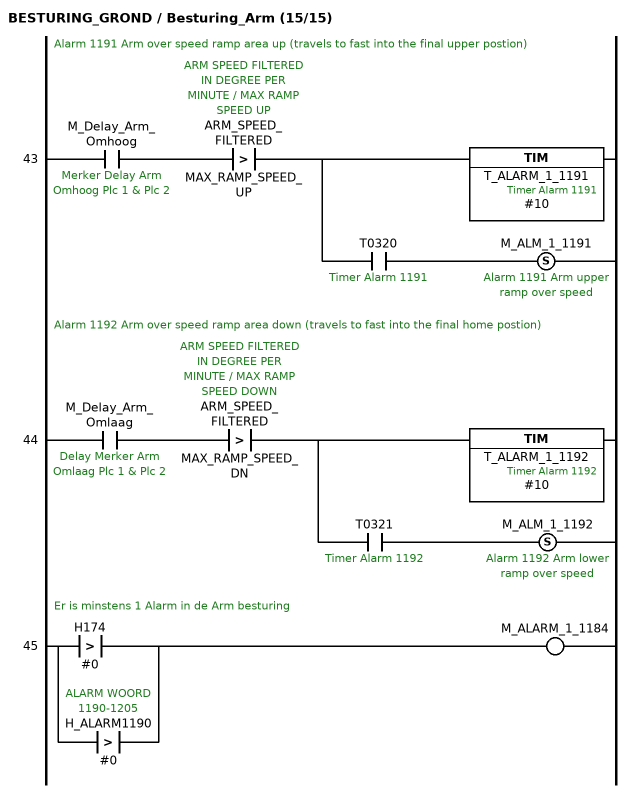
; [picture p168: BESTURING_GROND / Besturing_Arm, rungs 43-45]
; rung 43: Alarm 1191 Arm over speed ramp area up (travels to fast into the final upper postion)
LD M_Delay_Arm_Omhoog  ; Merker Delay Arm Omhoog Plc 1 & Plc 2
AND>F(333) ARM_SPEED_FILTERED MAX_RAMP_SPEED_UP  ; ARM SPEED FILTERED IN DEGREE PER MINUTE, MAX RAMP SPEED UP
TIM T_ALARM_1_1191 #10  ; Timer Alarm 1191
AND T0320  ; Timer Alarm 1191
SET M_ALM_1_1191  ; Alarm 1191 Arm upper ramp over speed
; rung 44: Alarm 1192 Arm over speed ramp area down (travels to fast into the final home postion)
LD M_Delay_Arm_Omlaag  ; Delay Merker Arm Omlaag Plc 1 & Plc 2
AND>F(333) ARM_SPEED_FILTERED MAX_RAMP_SPEED_DN  ; ARM SPEED FILTERED IN DEGREE PER MINUTE, MAX RAMP SPEED DOWN
TIM T_ALARM_1_1192 #10  ; Timer Alarm 1192
AND T0321  ; Timer Alarm 1192
SET M_ALM_1_1192  ; Alarm 1192 Arm lower ramp over speed
; rung 45: Er is minstens 1 Alarm in de Arm besturing
LD>(320) H174 #0
OR>(320) H_ALARM1190 #0  ; ALARM WOORD 1190-1205
OUT M_ALARM_1_1184

### Section Einde_Besturing_Grond
; rung 0
END(001)

## Program SIGNALEN_EILAND (cyclic task 10)

### Section Fast_Counter_Control
; rung 0: adress in 363-365 adrs uit 62-64

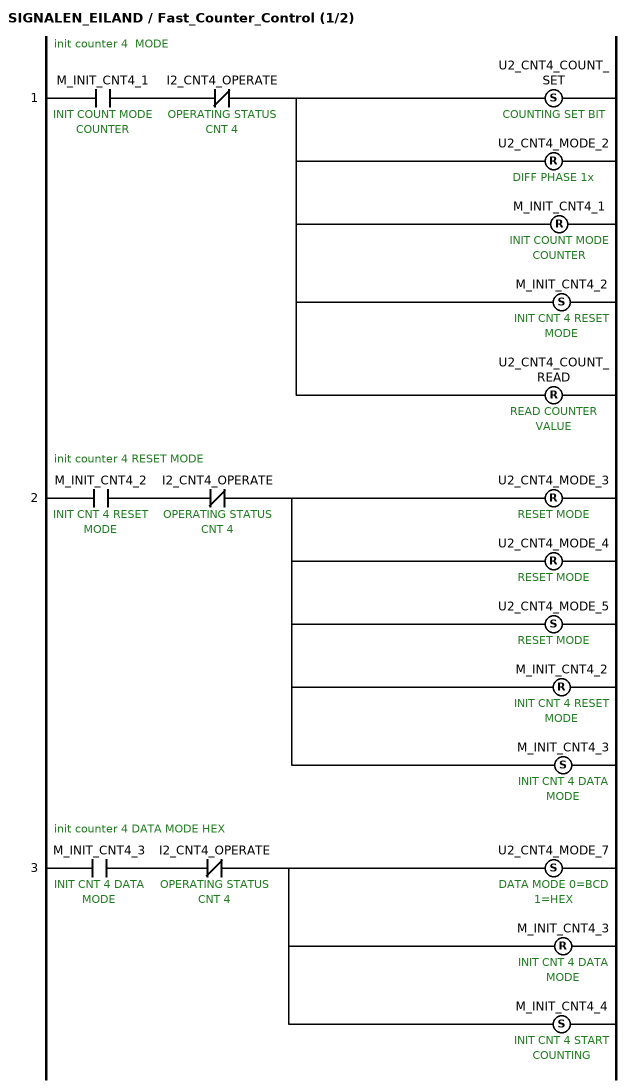
; rung 1: init counter 4  MODE
LD M_INIT_CNT4_1  ; INIT COUNT MODE COUNTER
ANDNOT I2_CNT4_OPERATE  ; OPERATING STATUS CNT 4
SET U2_CNT4_COUNT_SET  ; COUNTING SET BIT
RSET U2_CNT4_MODE_2  ; DIFF PHASE 1x
RSET M_INIT_CNT4_1  ; INIT COUNT MODE COUNTER
SET M_INIT_CNT4_2  ; INIT CNT 4 RESET MODE
RSET U2_CNT4_COUNT_READ  ; READ COUNTER VALUE
; rung 2: init counter 4 RESET MODE
LD M_INIT_CNT4_2  ; INIT CNT 4 RESET MODE
ANDNOT I2_CNT4_OPERATE  ; OPERATING STATUS CNT 4
RSET U2_CNT4_MODE_3  ; RESET MODE
RSET U2_CNT4_MODE_4  ; RESET MODE
SET U2_CNT4_MODE_5  ; RESET MODE
RSET M_INIT_CNT4_2  ; INIT CNT 4 RESET MODE
SET M_INIT_CNT4_3  ; INIT CNT 4 DATA MODE
; rung 3: init counter 4 DATA MODE HEX
LD M_INIT_CNT4_3  ; INIT CNT 4 DATA MODE
ANDNOT I2_CNT4_OPERATE  ; OPERATING STATUS CNT 4
SET U2_CNT4_MODE_7  ; DATA MODE 0=BCD 1=HEX
RSET M_INIT_CNT4_3  ; INIT CNT 4 DATA MODE
SET M_INIT_CNT4_4  ; INIT CNT 4 START COUNTING

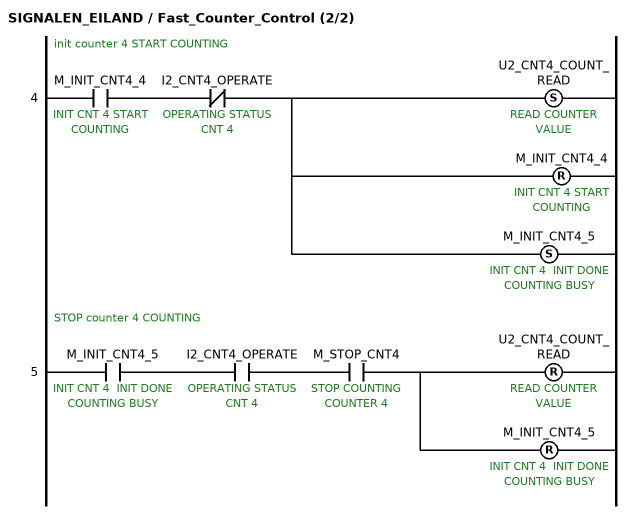
; rung 4: init counter 4 START COUNTING
LD M_INIT_CNT4_4  ; INIT CNT 4 START COUNTING
ANDNOT I2_CNT4_OPERATE  ; OPERATING STATUS CNT 4
SET U2_CNT4_COUNT_READ  ; READ COUNTER VALUE
RSET M_INIT_CNT4_4  ; INIT CNT 4 START COUNTING
SET M_INIT_CNT4_5  ; INIT CNT 4  INIT DONE COUNTING BUSY
; rung 5: STOP counter 4 COUNTING
LD M_INIT_CNT4_5  ; INIT CNT 4  INIT DONE COUNTING BUSY
AND I2_CNT4_OPERATE  ; OPERATING STATUS CNT 4
AND M_STOP_CNT4  ; STOP COUNTING COUNTER 4
RSET U2_CNT4_COUNT_READ  ; READ COUNTER VALUE
RSET M_INIT_CNT4_5  ; INIT CNT 4  INIT DONE COUNTING BUSY

### Section Incremental_Encoder_Decoder_4

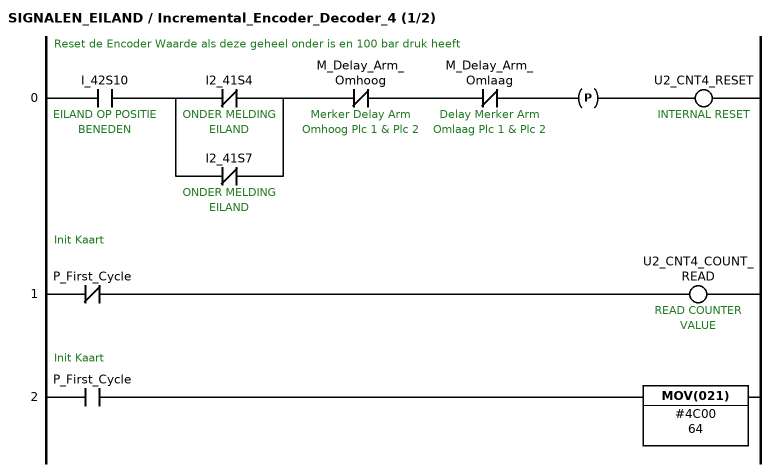
; rung 0: Reset de Encoder Waarde als deze geheel onder is en 100 bar druk heeft
LD I_42S10  ; EILAND OP POSITIE BENEDEN
LDNOT I2_41S4  ; ONDER MELDING EILAND
ORNOT I2_41S7  ; ONDER MELDING EILAND
ANDLD
ANDNOT M_Delay_Arm_Omhoog  ; Merker Delay Arm Omhoog Plc 1 & Plc 2
ANDNOT M_Delay_Arm_Omlaag  ; Delay Merker Arm Omlaag Plc 1 & Plc 2
UP(521)
OUT U2_CNT4_RESET  ; INTERNAL RESET
; rung 1: Init Kaart
LDNOT P_First_Cycle
OUT U2_CNT4_COUNT_READ  ; READ COUNTER VALUE
; rung 2: Init Kaart
LD P_First_Cycle
MOV(021) #4C00 64

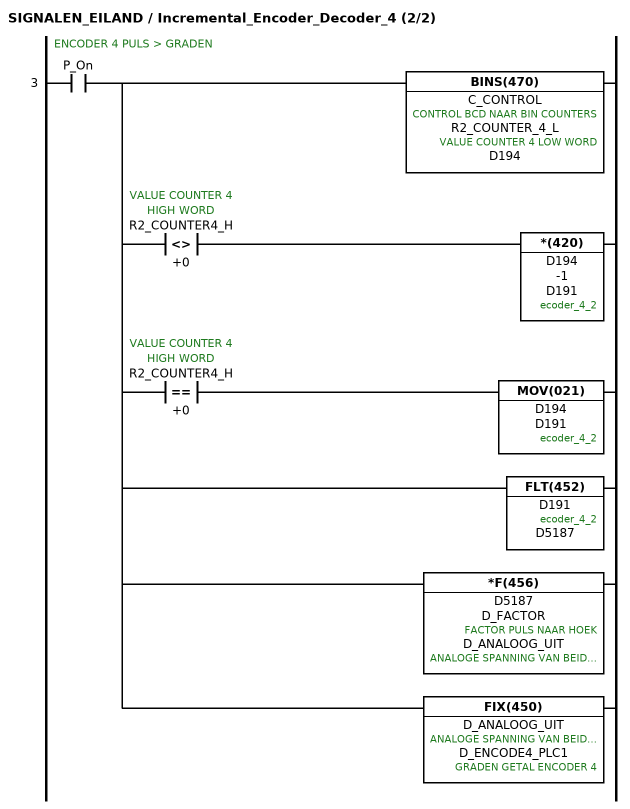
; rung 3: ENCODER 4 PULS > GRADEN
LD P_On
OUT TR0
BINS(470) C_CONTROL R2_COUNTER_4_L D194  ; CONTROL BCD NAAR BIN COUNTERS, VALUE COUNTER 4 LOW WORD
AND<>S(307) R2_COUNTER4_H +0  ; VALUE COUNTER 4 HIGH WORD
*(420) D194 -1 D191  ; ecoder_4_2
LD TR0
AND=S(302) R2_COUNTER4_H +0  ; VALUE COUNTER 4 HIGH WORD
MOV(021) D194 D191  ; ecoder_4_2
LD TR0
FLT(452) D191 D5187  ; ecoder_4_2
*F(456) D5187 D_FACTOR D_ANALOOG_UIT  ; FACTOR PULS NAAR HOEK, ANALOGE SPANNING VAN BEIDE PLC'S
FIX(450) D_ANALOOG_UIT D_ENCODE4_PLC1  ; ANALOGE SPANNING VAN BEIDE PLC'S, GRADEN GETAL ENCODER 4

### Section Horizon_Decoder_Eiland
; rung 0: De Horizon Decoder is alleen aanwezig in Plc 2 Omdat de analoog waarde allen daar binnen word gelezen.

### Section Controle_Positie_Eiland

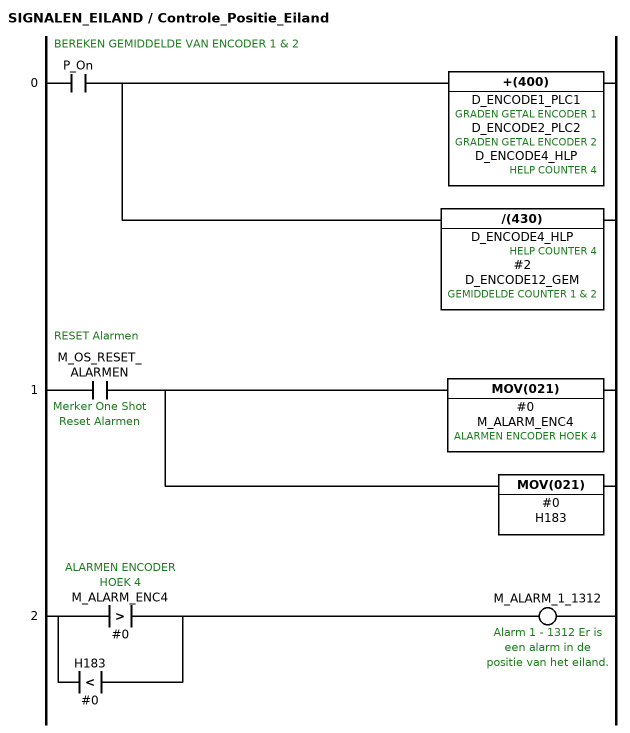
; rung 0: BEREKEN GEMIDDELDE VAN ENCODER 1 & 2
LD P_On
+(400) D_ENCODE1_PLC1 D_ENCODE2_PLC2 D_ENCODE4_HLP  ; GRADEN GETAL ENCODER 1, GRADEN GETAL ENCODER 2, HELP COUNTER 4
/(430) D_ENCODE4_HLP #2 D_ENCODE12_GEM  ; HELP COUNTER 4, GEMIDDELDE COUNTER 1 & 2
; rung 1: RESET Alarmen
LD M_OS_RESET_ALARMEN  ; Merker One Shot Reset Alarmen
MOV(021) #0 M_ALARM_ENC4  ; ALARMEN ENCODER HOEK 4
MOV(021) #0 H183
; rung 2
LD>(320) M_ALARM_ENC4 #0  ; ALARMEN ENCODER HOEK 4
OR<(310) H183 #0
OUT M_ALARM_1_1312  ; Alarm 1 - 1312 Er is een alarm in de positie van het eiland.

### Section Controle_Level_Switches_Eiland

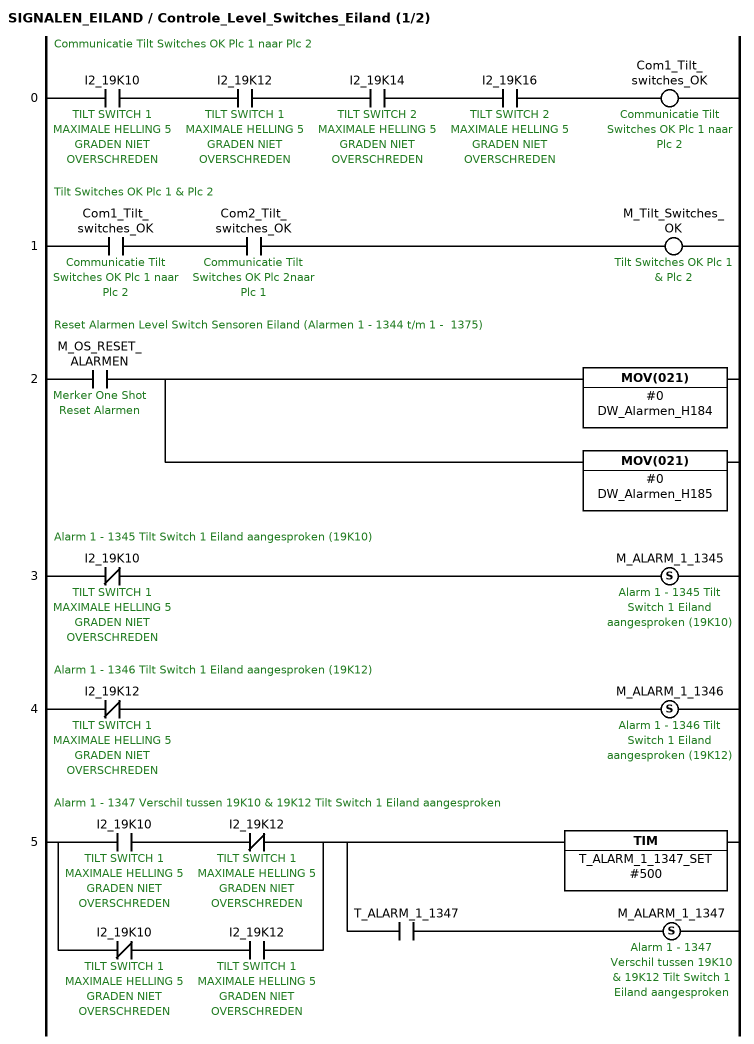
; rung 0: Communicatie Tilt Switches OK Plc 1 naar Plc 2
LD I2_19K10  ; TILT SWITCH 1 MAXIMALE HELLING 5 GRADEN NIET OVERSCHREDEN
AND I2_19K12  ; TILT SWITCH 1 MAXIMALE HELLING 5 GRADEN NIET OVERSCHREDEN
AND I2_19K14  ; TILT SWITCH 2 MAXIMALE HELLING 5 GRADEN NIET OVERSCHREDEN
AND I2_19K16  ; TILT SWITCH 2 MAXIMALE HELLING 5 GRADEN NIET OVERSCHREDEN
OUT Com1_Tilt_switches_OK  ; Communicatie Tilt Switches OK Plc 1 naar Plc 2
; rung 1: Tilt Switches OK Plc 1 & Plc 2
LD Com1_Tilt_switches_OK  ; Communicatie Tilt Switches OK Plc 1 naar Plc 2
AND Com2_Tilt_switches_OK  ; Communicatie Tilt Switches OK Plc 2naar Plc 1
OUT M_Tilt_Switches_OK  ; Tilt Switches OK Plc 1 & Plc 2
; rung 2: Reset Alarmen Level Switch Sensoren Eiland (Alarmen 1 - 1344 t/m 1 -  1375)
LD M_OS_RESET_ALARMEN  ; Merker One Shot Reset Alarmen
MOV(021) #0 DW_Alarmen_H184
MOV(021) #0 DW_Alarmen_H185
; rung 3: Alarm 1 - 1345 Tilt Switch 1 Eiland aangesproken (19K10)
LDNOT I2_19K10  ; TILT SWITCH 1 MAXIMALE HELLING 5 GRADEN NIET OVERSCHREDEN
SET M_ALARM_1_1345  ; Alarm 1 - 1345 Tilt Switch 1 Eiland aangesproken (19K10)
; rung 4: Alarm 1 - 1346 Tilt Switch 1 Eiland aangesproken (19K12)
LDNOT I2_19K12  ; TILT SWITCH 1 MAXIMALE HELLING 5 GRADEN NIET OVERSCHREDEN
SET M_ALARM_1_1346  ; Alarm 1 - 1346 Tilt Switch 1 Eiland aangesproken (19K12)
; rung 5: Alarm 1 - 1347 Verschil tussen 19K10 & 19K12 Tilt Switch 1 Eiland aangesproken
LD I2_19K10  ; TILT SWITCH 1 MAXIMALE HELLING 5 GRADEN NIET OVERSCHREDEN
ANDNOT I2_19K12  ; TILT SWITCH 1 MAXIMALE HELLING 5 GRADEN NIET OVERSCHREDEN
LDNOT I2_19K10  ; TILT SWITCH 1 MAXIMALE HELLING 5 GRADEN NIET OVERSCHREDEN
AND I2_19K12  ; TILT SWITCH 1 MAXIMALE HELLING 5 GRADEN NIET OVERSCHREDEN
ORLD
TIM T_ALARM_1_1347_SET #500
AND T_ALARM_1_1347
SET M_ALARM_1_1347  ; Alarm 1 - 1347 Verschil tussen 19K10 & 19K12 Tilt Switch 1 Eiland aangesproken

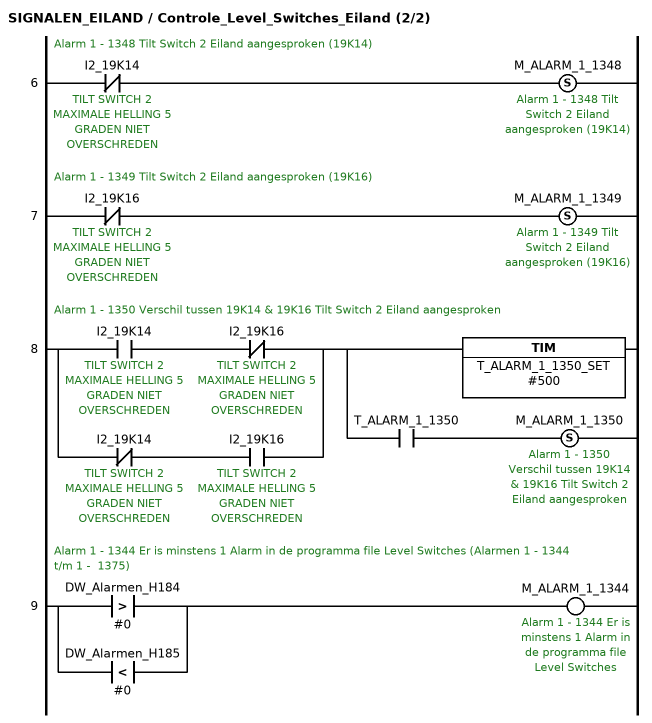
; rung 6: Alarm 1 - 1348 Tilt Switch 2 Eiland aangesproken (19K14)
LDNOT I2_19K14  ; TILT SWITCH 2 MAXIMALE HELLING 5 GRADEN NIET OVERSCHREDEN
SET M_ALARM_1_1348  ; Alarm 1 - 1348 Tilt Switch 2 Eiland aangesproken (19K14)
; rung 7: Alarm 1 - 1349 Tilt Switch 2 Eiland aangesproken (19K16)
LDNOT I2_19K16  ; TILT SWITCH 2 MAXIMALE HELLING 5 GRADEN NIET OVERSCHREDEN
SET M_ALARM_1_1349  ; Alarm 1 - 1349 Tilt Switch 2 Eiland aangesproken (19K16)
; rung 8: Alarm 1 - 1350 Verschil tussen 19K14 & 19K16 Tilt Switch 2 Eiland aangesproken
LD I2_19K14  ; TILT SWITCH 2 MAXIMALE HELLING 5 GRADEN NIET OVERSCHREDEN
ANDNOT I2_19K16  ; TILT SWITCH 2 MAXIMALE HELLING 5 GRADEN NIET OVERSCHREDEN
LDNOT I2_19K14  ; TILT SWITCH 2 MAXIMALE HELLING 5 GRADEN NIET OVERSCHREDEN
AND I2_19K16  ; TILT SWITCH 2 MAXIMALE HELLING 5 GRADEN NIET OVERSCHREDEN
ORLD
TIM T_ALARM_1_1350_SET #500
AND T_ALARM_1_1350
SET M_ALARM_1_1350  ; Alarm 1 - 1350 Verschil tussen 19K14 & 19K16 Tilt Switch 2 Eiland aangesproken
; rung 9: Alarm 1 - 1344 Er is minstens 1 Alarm in de programma file Level Switches (Alarmen 1 - 1344 t/m 1 -  1375)
LD>(320) DW_Alarmen_H184 #0
OR<(310) DW_Alarmen_H185 #0
OUT M_ALARM_1_1344  ; Alarm 1 - 1344 Er is minstens 1 Alarm in de programma file Level Switches

### Section Einde_Sinalering_Eiland
; rung 0
END(001)

## Program BESTURING_EILAND (cyclic task 11)
Local symbols
M_ALARM_1_1377 BOOL

### Section Poortjes_Eiland

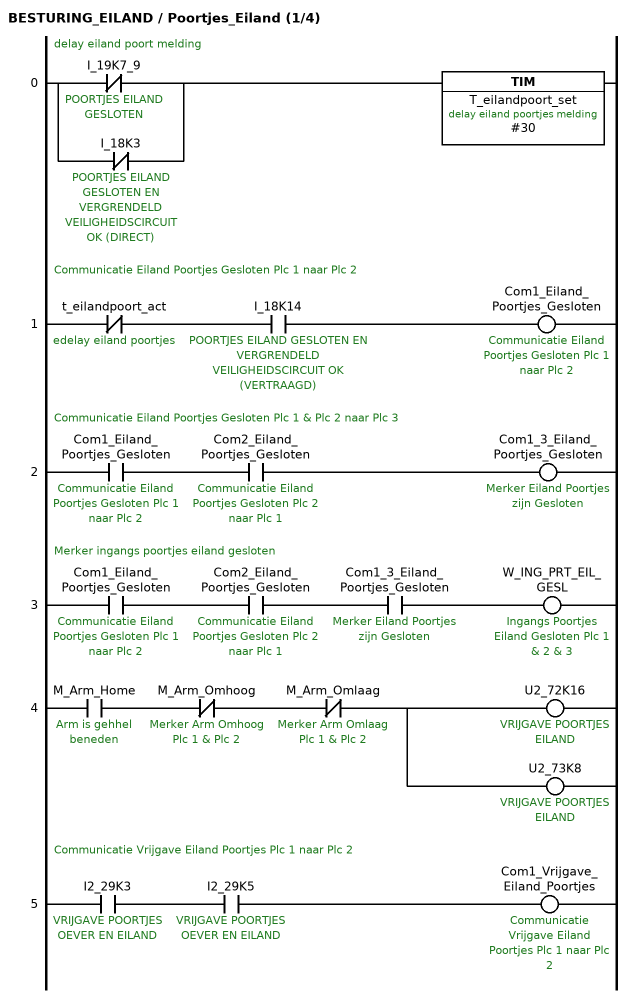
; rung 0: delay eiland poort melding
LDNOT I_19K7_9  ; POORTJES EILAND GESLOTEN
ORNOT I_18K3  ; POORTJES EILAND GESLOTEN EN VERGRENDELD VEILIGHEIDSCIRCUIT OK (DIRECT)
TIM T_eilandpoort_set #30  ; delay eiland poortjes melding
; rung 1: Communicatie Eiland Poortjes Gesloten Plc 1 naar Plc 2
LDNOT t_eilandpoort_act  ; edelay eiland poortjes
AND I_18K14  ; POORTJES EILAND GESLOTEN EN VERGRENDELD VEILIGHEIDSCIRCUIT OK (VERTRAAGD)
OUT Com1_Eiland_Poortjes_Gesloten  ; Communicatie Eiland Poortjes Gesloten Plc 1 naar Plc 2
; rung 2: Communicatie Eiland Poortjes Gesloten Plc 1 & Plc 2 naar Plc 3
LD Com1_Eiland_Poortjes_Gesloten  ; Communicatie Eiland Poortjes Gesloten Plc 1 naar Plc 2
AND Com2_Eiland_Poortjes_Gesloten  ; Communicatie Eiland Poortjes Gesloten Plc 2 naar Plc 1
OUT Com1_3_Eiland_Poortjes_Gesloten  ; Merker Eiland Poortjes zijn Gesloten
; rung 3: Merker ingangs poortjes eiland gesloten
LD Com1_Eiland_Poortjes_Gesloten  ; Communicatie Eiland Poortjes Gesloten Plc 1 naar Plc 2
AND Com2_Eiland_Poortjes_Gesloten  ; Communicatie Eiland Poortjes Gesloten Plc 2 naar Plc 1
AND Com1_3_Eiland_Poortjes_Gesloten  ; Merker Eiland Poortjes zijn Gesloten
OUT W_ING_PRT_EIL_GESL  ; Ingangs Poortjes Eiland Gesloten Plc 1 & 2 & 3
; rung 4
LD M_Arm_Home  ; Arm is gehhel beneden
ANDNOT M_Arm_Omhoog  ; Merker Arm Omhoog Plc 1 & Plc 2
ANDNOT M_Arm_Omlaag  ; Merker Arm Omlaag Plc 1 & Plc 2
OUT U2_72K16  ; VRIJGAVE POORTJES EILAND
OUT U2_73K8  ; VRIJGAVE POORTJES EILAND
; rung 5: Communicatie Vrijgave Eiland Poortjes Plc 1 naar Plc 2
LD I2_29K3  ; VRIJGAVE POORTJES OEVER EN EILAND
AND I2_29K5  ; VRIJGAVE POORTJES OEVER EN EILAND
OUT Com1_Vrijgave_Eiland_Poortjes  ; Communicatie Vrijgave Eiland Poortjes Plc 1 naar Plc 2

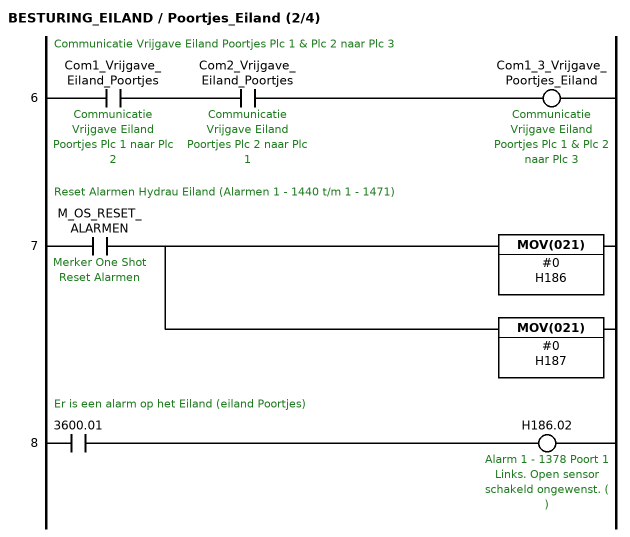
; rung 6: Communicatie Vrijgave Eiland Poortjes Plc 1 & Plc 2 naar Plc 3
LD Com1_Vrijgave_Eiland_Poortjes  ; Communicatie Vrijgave Eiland Poortjes Plc 1 naar Plc 2
AND Com2_Vrijgave_Eiland_Poortjes  ; Communicatie Vrijgave Eiland Poortjes Plc 2 naar Plc 1
OUT Com1_3_Vrijgave_Poortjes_Eiland  ; Communicatie Vrijgave Eiland Poortjes Plc 1 & Plc 2 naar Plc 3
; rung 7: Reset Alarmen Hydrau Eiland (Alarmen 1 - 1440 t/m 1 - 1471)
LD M_OS_RESET_ALARMEN  ; Merker One Shot Reset Alarmen
MOV(021) #0 H186
MOV(021) #0 H187
; rung 8: Er is een alarm op het Eiland (eiland Poortjes)
LD 3600.01
OUT H186.02  ; Alarm 1 - 1378 Poort 1 Links. Open sensor schakeld ongewenst. ( )

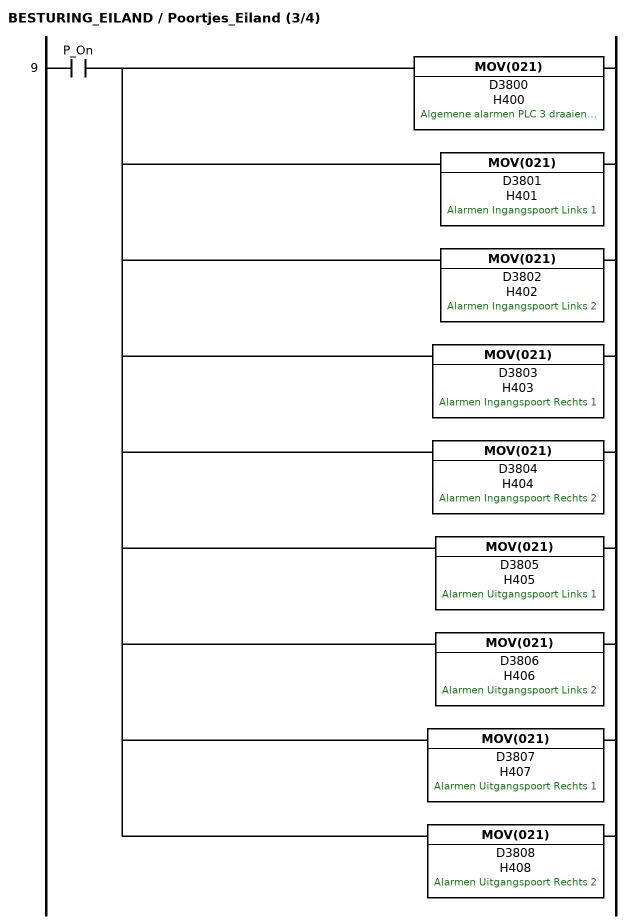
; rung 9
LD P_On
MOV(021) D3800 H400  ; Algemene alarmen PLC 3 draaiend deel eiland
MOV(021) D3801 H401  ; Alarmen Ingangspoort Links 1
MOV(021) D3802 H402  ; Alarmen Ingangspoort Links 2
MOV(021) D3803 H403  ; Alarmen Ingangspoort Rechts 1
MOV(021) D3804 H404  ; Alarmen Ingangspoort Rechts 2
MOV(021) D3805 H405  ; Alarmen Uitgangspoort Links 1
MOV(021) D3806 H406  ; Alarmen Uitgangspoort Links 2
MOV(021) D3807 H407  ; Alarmen Uitgangspoort Rechts 1
MOV(021) D3808 H408  ; Alarmen Uitgangspoort Rechts 2

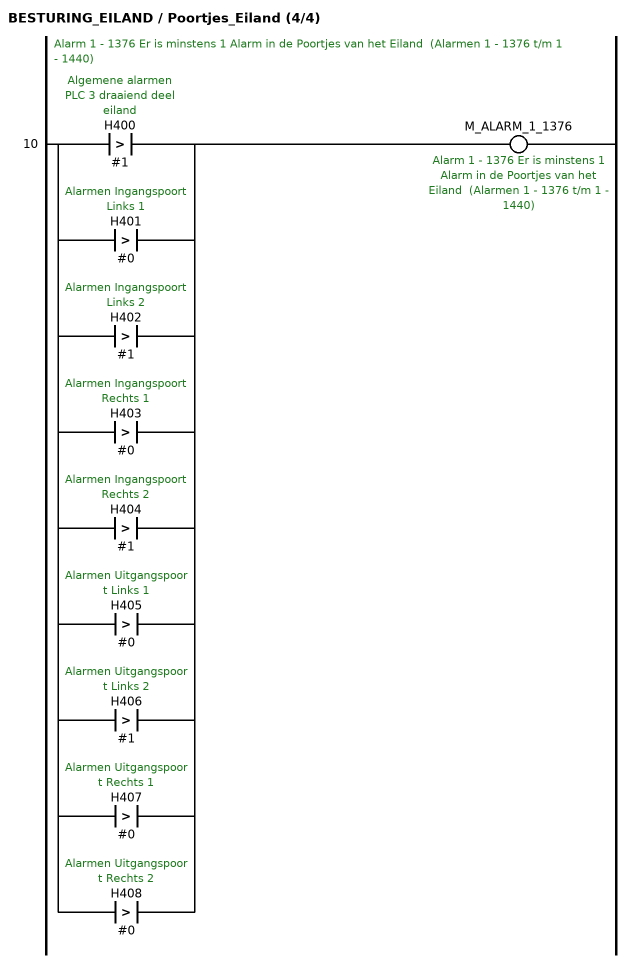
; rung 10: Alarm 1 - 1376 Er is minstens 1 Alarm in de Poortjes van het Eiland  (Alarmen 1 - 1376 t/m 1 - 1440)
LD>(320) H400 #1  ; Algemene alarmen PLC 3 draaiend deel eiland
OR>(320) H401 #0  ; Alarmen Ingangspoort Links 1
OR>(320) H402 #1  ; Alarmen Ingangspoort Links 2
OR>(320) H403 #0  ; Alarmen Ingangspoort Rechts 1
OR>(320) H404 #1  ; Alarmen Ingangspoort Rechts 2
OR>(320) H405 #0  ; Alarmen Uitgangspoort Links 1
OR>(320) H406 #1  ; Alarmen Uitgangspoort Links 2
OR>(320) H407 #0  ; Alarmen Uitgangspoort Rechts 1
OR>(320) H408 #0  ; Alarmen Uitgangspoort Rechts 2
OUT M_ALARM_1_1376  ; Alarm 1 - 1376 Er is minstens 1 Alarm in de Poortjes van het Eiland  (Alarmen 1 - 1376 t/m 1 - 1440)

### Section Hydrauliek_Eiland

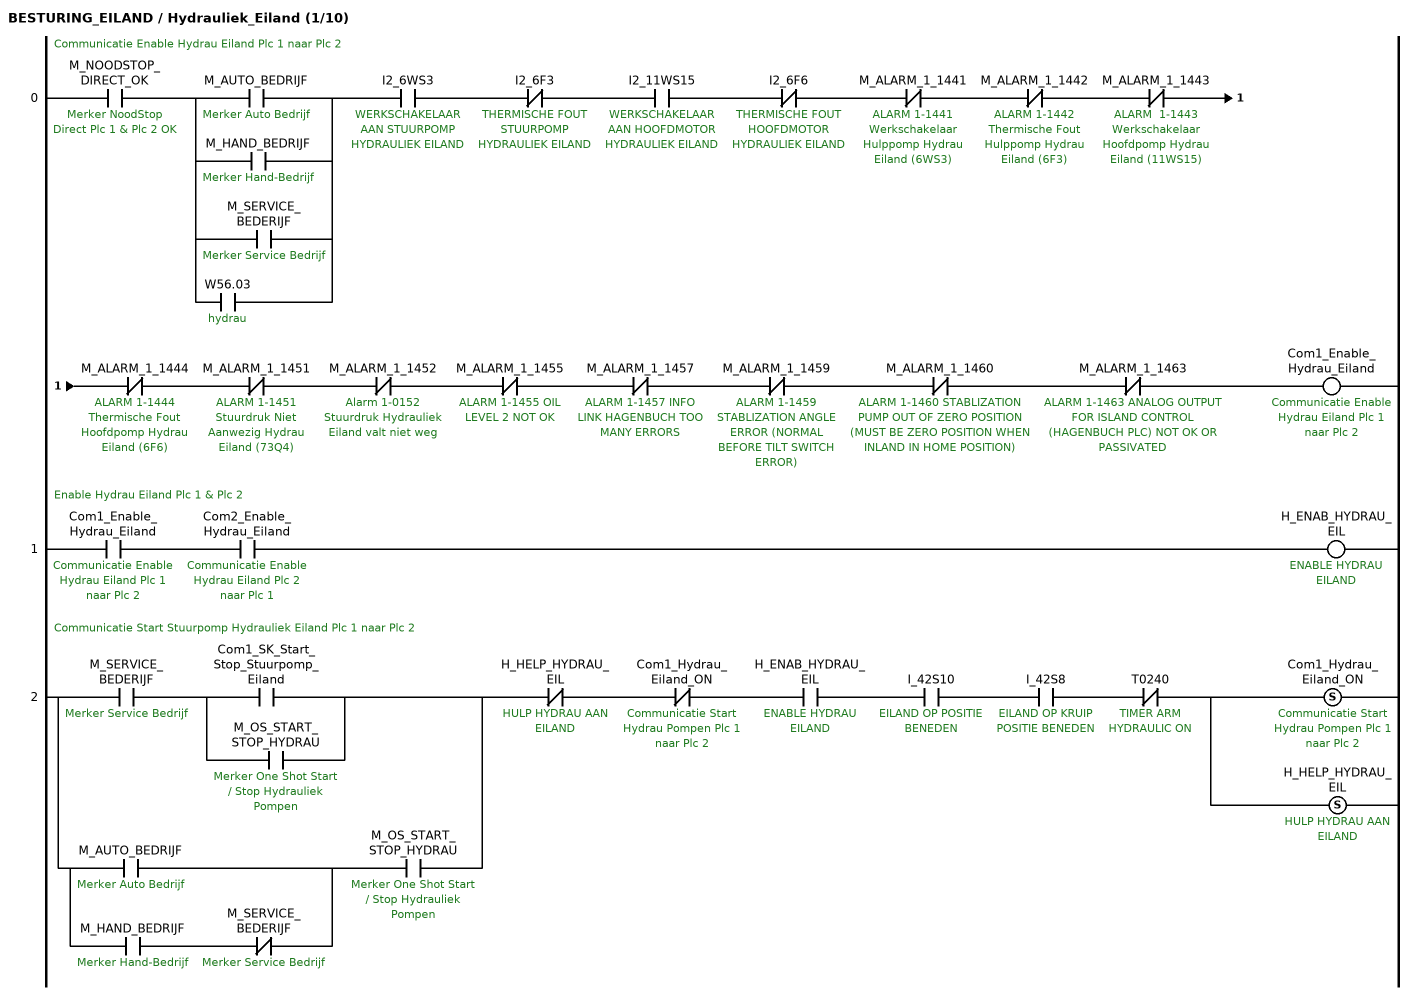
; rung 0: Communicatie Enable Hydrau Eiland Plc 1 naar Plc 2
LD M_NOODSTOP_DIRECT_OK  ; Merker NoodStop Direct Plc 1 & Plc 2 OK
LD M_AUTO_BEDRIJF  ; Merker Auto Bedrijf
OR M_HAND_BEDRIJF  ; Merker Hand-Bedrijf
OR M_SERVICE_BEDERIJF  ; Merker Service Bedrijf
OR W56.03  ; hydrau
ANDLD
AND I2_6WS3  ; WERKSCHAKELAAR AAN STUURPOMP HYDRAULIEK EILAND
ANDNOT I2_6F3  ; THERMISCHE FOUT STUURPOMP HYDRAULIEK EILAND
AND I2_11WS15  ; WERKSCHAKELAAR AAN HOOFDMOTOR HYDRAULIEK EILAND
ANDNOT I2_6F6  ; THERMISCHE FOUT HOOFDMOTOR HYDRAULIEK EILAND
ANDNOT M_ALARM_1_1441  ; ALARM 1-1441 Werkschakelaar Hulppomp Hydrau Eiland (6WS3)
ANDNOT M_ALARM_1_1442  ; ALARM 1-1442 Thermische Fout Hulppomp Hydrau Eiland (6F3)
ANDNOT M_ALARM_1_1443  ; ALARM  1-1443 Werkschakelaar Hoofdpomp Hydrau Eiland (11WS15)
ANDNOT M_ALARM_1_1444  ; ALARM 1-1444 Thermische Fout Hoofdpomp Hydrau Eiland (6F6)
ANDNOT M_ALARM_1_1451  ; ALARM 1-1451 Stuurdruk Niet Aanwezig Hydrau Eiland (73Q4)
ANDNOT M_ALARM_1_1452  ; Alarm 1-0152 Stuurdruk Hydrauliek Eiland valt niet weg
ANDNOT M_ALARM_1_1455  ; ALARM 1-1455 OIL LEVEL 2 NOT OK
ANDNOT M_ALARM_1_1457  ; ALARM 1-1457 INFO LINK HAGENBUCH TOO MANY ERRORS
ANDNOT M_ALARM_1_1459  ; ALARM 1-1459 STABLIZATION ANGLE ERROR (NORMAL BEFORE TILT SWITCH ERROR)
ANDNOT M_ALARM_1_1460  ; ALARM 1-1460 STABLIZATION PUMP OUT OF ZERO POSITION (MUST BE ZERO POSITION WHEN INLAND IN HOME POSITION)
ANDNOT M_ALARM_1_1463  ; ALARM 1-1463 ANALOG OUTPUT FOR ISLAND CONTROL (HAGENBUCH PLC) NOT OK OR PASSIVATED
OUT Com1_Enable_Hydrau_Eiland  ; Communicatie Enable Hydrau Eiland Plc 1 naar Plc 2
; rung 1: Enable Hydrau Eiland Plc 1 & Plc 2
LD Com1_Enable_Hydrau_Eiland  ; Communicatie Enable Hydrau Eiland Plc 1 naar Plc 2
AND Com2_Enable_Hydrau_Eiland  ; Communicatie Enable Hydrau Eiland Plc 2 naar Plc 1
OUT H_ENAB_HYDRAU_EIL  ; ENABLE HYDRAU EILAND
; rung 2: Communicatie Start Stuurpomp Hydrauliek Eiland Plc 1 naar Plc 2
LD M_SERVICE_BEDERIJF  ; Merker Service Bedrijf
LD Com1_SK_Start_Stop_Stuurpomp_Eiland
OR M_OS_START_STOP_HYDRAU  ; Merker One Shot Start / Stop Hydrauliek Pompen
ANDLD
LD M_AUTO_BEDRIJF  ; Merker Auto Bedrijf
LD M_HAND_BEDRIJF  ; Merker Hand-Bedrijf
ANDNOT M_SERVICE_BEDERIJF  ; Merker Service Bedrijf
ORLD
AND M_OS_START_STOP_HYDRAU  ; Merker One Shot Start / Stop Hydrauliek Pompen
ORLD
ANDNOT H_HELP_HYDRAU_EIL  ; HULP HYDRAU AAN EILAND
ANDNOT Com1_Hydrau_Eiland_ON  ; Communicatie Start Hydrau Pompen Plc 1 naar Plc 2
AND H_ENAB_HYDRAU_EIL  ; ENABLE HYDRAU EILAND
AND I_42S10  ; EILAND OP POSITIE BENEDEN
AND I_42S8  ; EILAND OP KRUIP POSITIE BENEDEN
ANDNOT T0240  ; TIMER ARM HYDRAULIC ON
SET Com1_Hydrau_Eiland_ON  ; Communicatie Start Hydrau Pompen Plc 1 naar Plc 2
SET H_HELP_HYDRAU_EIL  ; HULP HYDRAU AAN EILAND

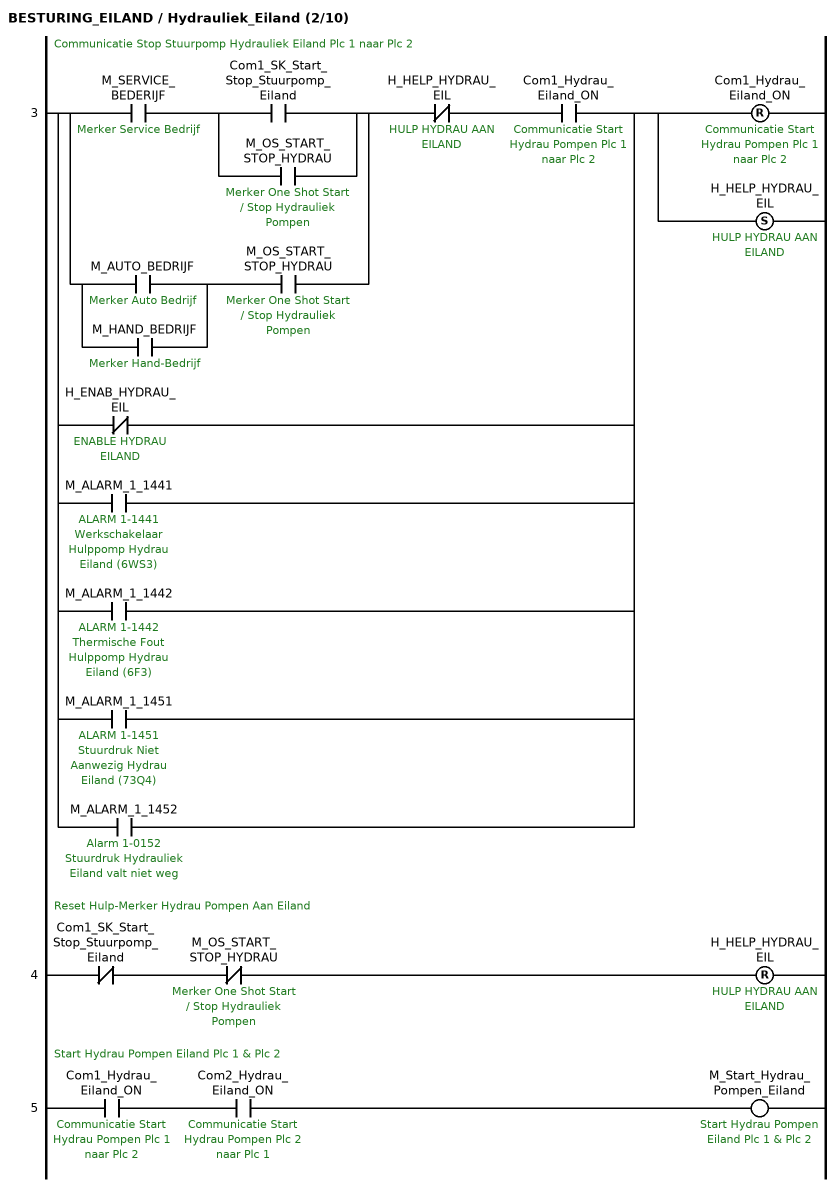
; rung 3: Communicatie Stop Stuurpomp Hydrauliek Eiland Plc 1 naar Plc 2
LD M_SERVICE_BEDERIJF  ; Merker Service Bedrijf
LD Com1_SK_Start_Stop_Stuurpomp_Eiland
OR M_OS_START_STOP_HYDRAU  ; Merker One Shot Start / Stop Hydrauliek Pompen
ANDLD
LD M_AUTO_BEDRIJF  ; Merker Auto Bedrijf
OR M_HAND_BEDRIJF  ; Merker Hand-Bedrijf
AND M_OS_START_STOP_HYDRAU  ; Merker One Shot Start / Stop Hydrauliek Pompen
ORLD
ANDNOT H_HELP_HYDRAU_EIL  ; HULP HYDRAU AAN EILAND
AND Com1_Hydrau_Eiland_ON  ; Communicatie Start Hydrau Pompen Plc 1 naar Plc 2
ORNOT H_ENAB_HYDRAU_EIL  ; ENABLE HYDRAU EILAND
OR M_ALARM_1_1441  ; ALARM 1-1441 Werkschakelaar Hulppomp Hydrau Eiland (6WS3)
OR M_ALARM_1_1442  ; ALARM 1-1442 Thermische Fout Hulppomp Hydrau Eiland (6F3)
OR M_ALARM_1_1451  ; ALARM 1-1451 Stuurdruk Niet Aanwezig Hydrau Eiland (73Q4)
OR M_ALARM_1_1452  ; Alarm 1-0152 Stuurdruk Hydrauliek Eiland valt niet weg
RSET Com1_Hydrau_Eiland_ON  ; Communicatie Start Hydrau Pompen Plc 1 naar Plc 2
SET H_HELP_HYDRAU_EIL  ; HULP HYDRAU AAN EILAND
; rung 4: Reset Hulp-Merker Hydrau Pompen Aan Eiland
LDNOT Com1_SK_Start_Stop_Stuurpomp_Eiland
ANDNOT M_OS_START_STOP_HYDRAU  ; Merker One Shot Start / Stop Hydrauliek Pompen
RSET H_HELP_HYDRAU_EIL  ; HULP HYDRAU AAN EILAND
; rung 5: Start Hydrau Pompen Eiland Plc 1 & Plc 2
LD Com1_Hydrau_Eiland_ON  ; Communicatie Start Hydrau Pompen Plc 1 naar Plc 2
AND Com2_Hydrau_Eiland_ON  ; Communicatie Start Hydrau Pompen Plc 2 naar Plc 1
OUT M_Start_Hydrau_Pompen_Eiland  ; Start Hydrau Pompen Eiland Plc 1 & Plc 2

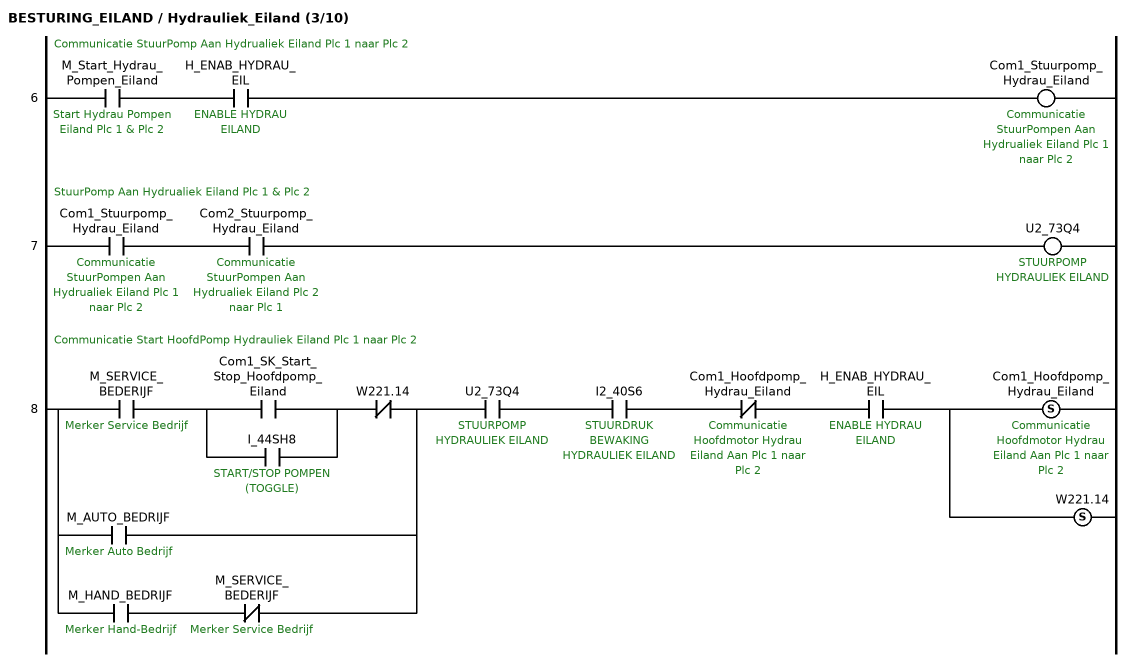
; rung 6: Communicatie StuurPomp Aan Hydrualiek Eiland Plc 1 naar Plc 2
LD M_Start_Hydrau_Pompen_Eiland  ; Start Hydrau Pompen Eiland Plc 1 & Plc 2
AND H_ENAB_HYDRAU_EIL  ; ENABLE HYDRAU EILAND
OUT Com1_Stuurpomp_Hydrau_Eiland  ; Communicatie StuurPompen Aan Hydrualiek Eiland Plc 1 naar Plc 2
; rung 7: StuurPomp Aan Hydrualiek Eiland Plc 1 & Plc 2
LD Com1_Stuurpomp_Hydrau_Eiland  ; Communicatie StuurPompen Aan Hydrualiek Eiland Plc 1 naar Plc 2
AND Com2_Stuurpomp_Hydrau_Eiland  ; Communicatie StuurPompen Aan Hydrualiek Eiland Plc 2 naar Plc 1
OUT U2_73Q4  ; STUURPOMP HYDRAULIEK EILAND
; rung 8: Communicatie Start HoofdPomp Hydrauliek Eiland Plc 1 naar Plc 2
LD M_SERVICE_BEDERIJF  ; Merker Service Bedrijf
LD Com1_SK_Start_Stop_Hoofdpomp_Eiland
OR I_44SH8  ; START/STOP POMPEN (TOGGLE)
ANDLD
ANDNOT W221.14
OR M_AUTO_BEDRIJF  ; Merker Auto Bedrijf
LD M_HAND_BEDRIJF  ; Merker Hand-Bedrijf
ANDNOT M_SERVICE_BEDERIJF  ; Merker Service Bedrijf
ORLD
AND U2_73Q4  ; STUURPOMP HYDRAULIEK EILAND
AND I2_40S6  ; STUURDRUK BEWAKING HYDRAULIEK EILAND
ANDNOT Com1_Hoofdpomp_Hydrau_Eiland  ; Communicatie Hoofdmotor Hydrau Eiland Aan Plc 1 naar Plc 2
AND H_ENAB_HYDRAU_EIL  ; ENABLE HYDRAU EILAND
SET Com1_Hoofdpomp_Hydrau_Eiland  ; Communicatie Hoofdmotor Hydrau Eiland Aan Plc 1 naar Plc 2
SET W221.14

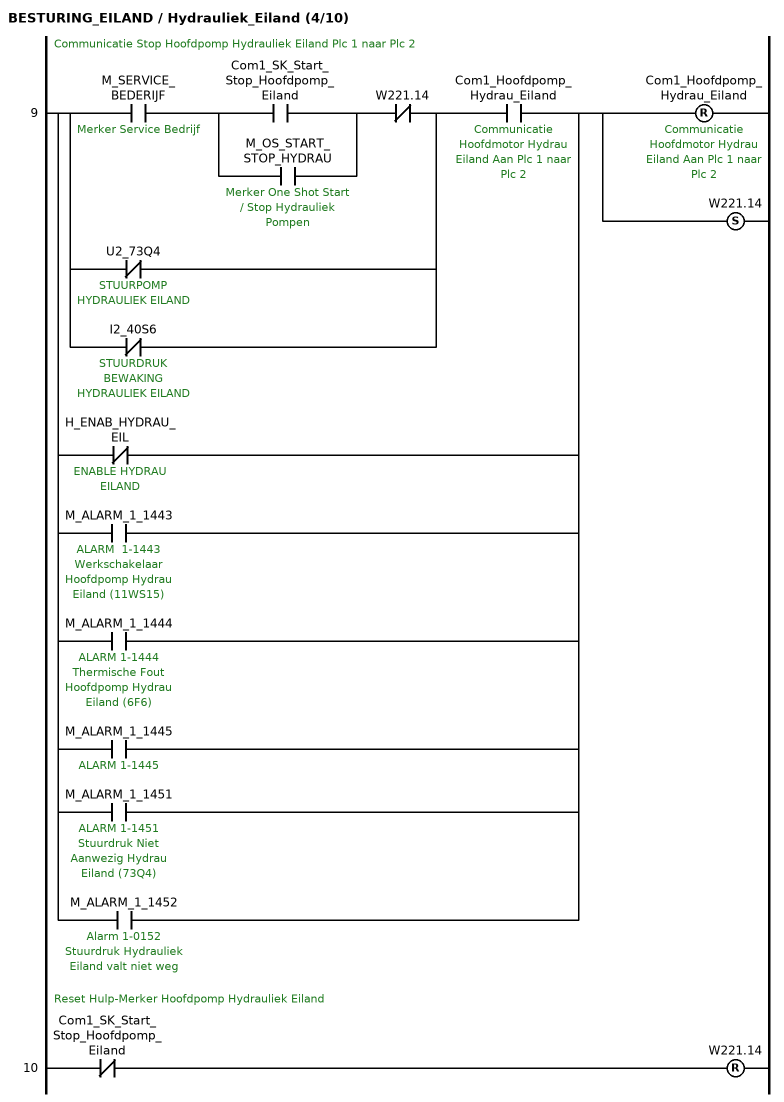
; rung 9: Communicatie Stop Hoofdpomp Hydrauliek Eiland Plc 1 naar Plc 2
LD M_SERVICE_BEDERIJF  ; Merker Service Bedrijf
LD Com1_SK_Start_Stop_Hoofdpomp_Eiland
OR M_OS_START_STOP_HYDRAU  ; Merker One Shot Start / Stop Hydrauliek Pompen
ANDLD
ANDNOT W221.14
ORNOT U2_73Q4  ; STUURPOMP HYDRAULIEK EILAND
ORNOT I2_40S6  ; STUURDRUK BEWAKING HYDRAULIEK EILAND
AND Com1_Hoofdpomp_Hydrau_Eiland  ; Communicatie Hoofdmotor Hydrau Eiland Aan Plc 1 naar Plc 2
ORNOT H_ENAB_HYDRAU_EIL  ; ENABLE HYDRAU EILAND
OR M_ALARM_1_1443  ; ALARM  1-1443 Werkschakelaar Hoofdpomp Hydrau Eiland (11WS15)
OR M_ALARM_1_1444  ; ALARM 1-1444 Thermische Fout Hoofdpomp Hydrau Eiland (6F6)
OR M_ALARM_1_1445  ; ALARM 1-1445
OR M_ALARM_1_1451  ; ALARM 1-1451 Stuurdruk Niet Aanwezig Hydrau Eiland (73Q4)
OR M_ALARM_1_1452  ; Alarm 1-0152 Stuurdruk Hydrauliek Eiland valt niet weg
RSET Com1_Hoofdpomp_Hydrau_Eiland  ; Communicatie Hoofdmotor Hydrau Eiland Aan Plc 1 naar Plc 2
SET W221.14
; rung 10: Reset Hulp-Merker Hoofdpomp Hydrauliek Eiland
LDNOT Com1_SK_Start_Stop_Hoofdpomp_Eiland
RSET W221.14

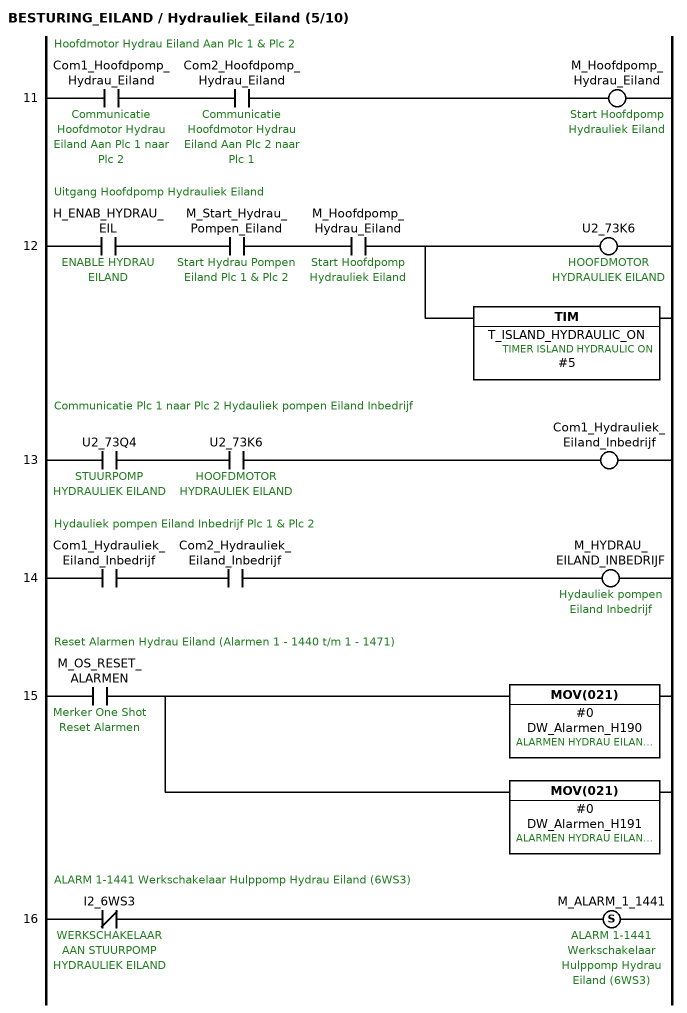
; rung 11: Hoofdmotor Hydrau Eiland Aan Plc 1 & Plc 2
LD Com1_Hoofdpomp_Hydrau_Eiland  ; Communicatie Hoofdmotor Hydrau Eiland Aan Plc 1 naar Plc 2
AND Com2_Hoofdpomp_Hydrau_Eiland  ; Communicatie Hoofdmotor Hydrau Eiland Aan Plc 2 naar Plc 1
OUT M_Hoofdpomp_Hydrau_Eiland  ; Start Hoofdpomp Hydrauliek Eiland
; rung 12: Uitgang Hoofdpomp Hydrauliek Eiland
LD H_ENAB_HYDRAU_EIL  ; ENABLE HYDRAU EILAND
AND M_Start_Hydrau_Pompen_Eiland  ; Start Hydrau Pompen Eiland Plc 1 & Plc 2
AND M_Hoofdpomp_Hydrau_Eiland  ; Start Hoofdpomp Hydrauliek Eiland
OUT U2_73K6  ; HOOFDMOTOR HYDRAULIEK EILAND
TIM T_ISLAND_HYDRAULIC_ON #5  ; TIMER ISLAND HYDRAULIC ON
; rung 13: Communicatie Plc 1 naar Plc 2 Hydauliek pompen Eiland Inbedrijf
LD U2_73Q4  ; STUURPOMP HYDRAULIEK EILAND
AND U2_73K6  ; HOOFDMOTOR HYDRAULIEK EILAND
OUT Com1_Hydrauliek_Eiland_Inbedrijf
; rung 14: Hydauliek pompen Eiland Inbedrijf Plc 1 & Plc 2
LD Com1_Hydrauliek_Eiland_Inbedrijf
AND Com2_Hydrauliek_Eiland_Inbedrijf
OUT M_HYDRAU_EILAND_INBEDRIJF  ; Hydauliek pompen Eiland Inbedrijf
; rung 15: Reset Alarmen Hydrau Eiland (Alarmen 1 - 1440 t/m 1 - 1471)
LD M_OS_RESET_ALARMEN  ; Merker One Shot Reset Alarmen
MOV(021) #0 DW_Alarmen_H190  ; ALARMEN HYDRAU EILAND 1440-1455
MOV(021) #0 DW_Alarmen_H191  ; ALARMEN HYDRAU EILAND 1456-1471
; rung 16: ALARM 1-1441 Werkschakelaar Hulppomp Hydrau Eiland (6WS3)
LDNOT I2_6WS3  ; WERKSCHAKELAAR AAN STUURPOMP HYDRAULIEK EILAND
SET M_ALARM_1_1441  ; ALARM 1-1441 Werkschakelaar Hulppomp Hydrau Eiland (6WS3)

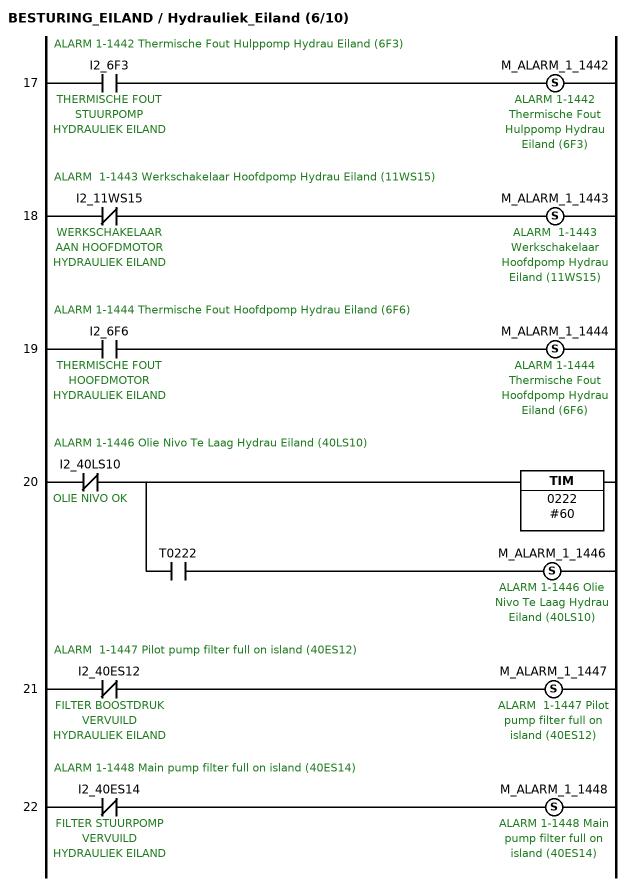
; rung 17: ALARM 1-1442 Thermische Fout Hulppomp Hydrau Eiland (6F3)
LD I2_6F3  ; THERMISCHE FOUT STUURPOMP HYDRAULIEK EILAND
SET M_ALARM_1_1442  ; ALARM 1-1442 Thermische Fout Hulppomp Hydrau Eiland (6F3)
; rung 18: ALARM  1-1443 Werkschakelaar Hoofdpomp Hydrau Eiland (11WS15)
LDNOT I2_11WS15  ; WERKSCHAKELAAR AAN HOOFDMOTOR HYDRAULIEK EILAND
SET M_ALARM_1_1443  ; ALARM  1-1443 Werkschakelaar Hoofdpomp Hydrau Eiland (11WS15)
; rung 19: ALARM 1-1444 Thermische Fout Hoofdpomp Hydrau Eiland (6F6)
LD I2_6F6  ; THERMISCHE FOUT HOOFDMOTOR HYDRAULIEK EILAND
SET M_ALARM_1_1444  ; ALARM 1-1444 Thermische Fout Hoofdpomp Hydrau Eiland (6F6)
; rung 20: ALARM 1-1446 Olie Nivo Te Laag Hydrau Eiland (40LS10)
LDNOT I2_40LS10  ; OLIE NIVO OK
TIM 0222 #60
AND T0222
SET M_ALARM_1_1446  ; ALARM 1-1446 Olie Nivo Te Laag Hydrau Eiland (40LS10)
; rung 21: ALARM  1-1447 Pilot pump filter full on island (40ES12)
LDNOT I2_40ES12  ; FILTER BOOSTDRUK VERVUILD HYDRAULIEK EILAND
SET M_ALARM_1_1447  ; ALARM  1-1447 Pilot pump filter full on island (40ES12)
; rung 22: ALARM 1-1448 Main pump filter full on island (40ES14)
LDNOT I2_40ES14  ; FILTER STUURPOMP VERVUILD HYDRAULIEK EILAND
SET M_ALARM_1_1448  ; ALARM 1-1448 Main pump filter full on island (40ES14)

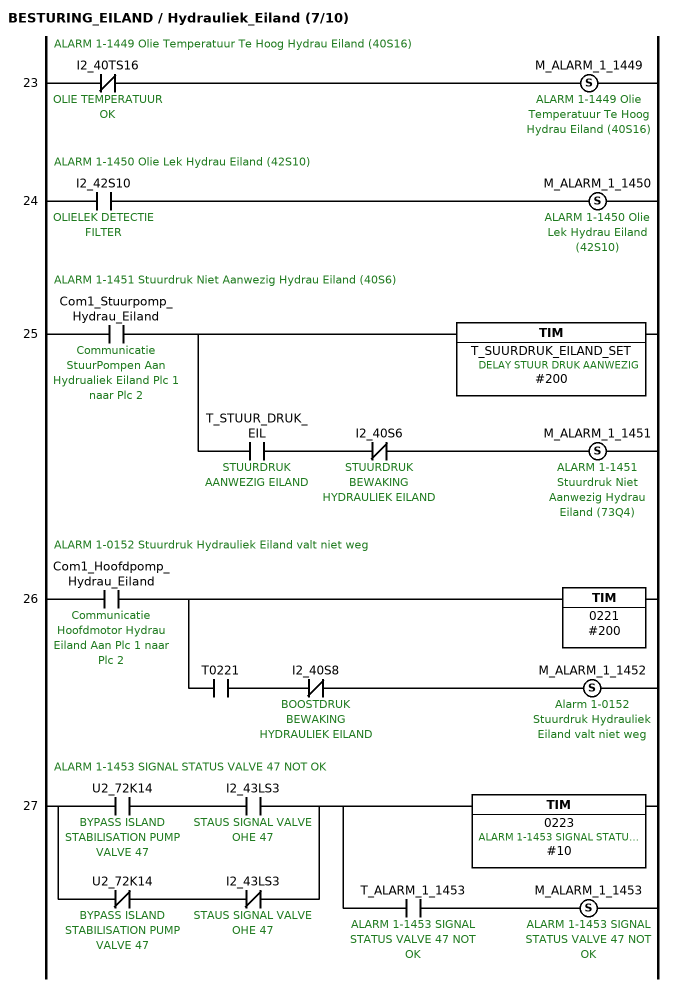
; rung 23: ALARM 1-1449 Olie Temperatuur Te Hoog Hydrau Eiland (40S16)
LDNOT I2_40TS16  ; OLIE TEMPERATUUR OK
SET M_ALARM_1_1449  ; ALARM 1-1449 Olie Temperatuur Te Hoog Hydrau Eiland (40S16)
; rung 24: ALARM 1-1450 Olie Lek Hydrau Eiland (42S10)
LD I2_42S10  ; OLIELEK DETECTIE FILTER
SET M_ALARM_1_1450  ; ALARM 1-1450 Olie Lek Hydrau Eiland (42S10)
; rung 25: ALARM 1-1451 Stuurdruk Niet Aanwezig Hydrau Eiland (40S6)
LD Com1_Stuurpomp_Hydrau_Eiland  ; Communicatie StuurPompen Aan Hydrualiek Eiland Plc 1 naar Plc 2
TIM T_SUURDRUK_EILAND_SET #200  ; DELAY STUUR DRUK AANWEZIG
AND T_STUUR_DRUK_EIL  ; STUURDRUK AANWEZIG EILAND
ANDNOT I2_40S6  ; STUURDRUK BEWAKING HYDRAULIEK EILAND
SET M_ALARM_1_1451  ; ALARM 1-1451 Stuurdruk Niet Aanwezig Hydrau Eiland (73Q4)
; rung 26: ALARM 1-0152 Stuurdruk Hydrauliek Eiland valt niet weg
LD Com1_Hoofdpomp_Hydrau_Eiland  ; Communicatie Hoofdmotor Hydrau Eiland Aan Plc 1 naar Plc 2
TIM 0221 #200
AND T0221
ANDNOT I2_40S8  ; BOOSTDRUK BEWAKING HYDRAULIEK EILAND
SET M_ALARM_1_1452  ; Alarm 1-0152 Stuurdruk Hydrauliek Eiland valt niet weg
; rung 27: ALARM 1-1453 SIGNAL STATUS VALVE 47 NOT OK
LD U2_72K14  ; BYPASS ISLAND STABILISATION PUMP VALVE 47
AND I2_43LS3  ; STAUS SIGNAL VALVE OHE 47
LDNOT U2_72K14  ; BYPASS ISLAND STABILISATION PUMP VALVE 47
ANDNOT I2_43LS3  ; STAUS SIGNAL VALVE OHE 47
ORLD
TIM 0223 #10  ; ALARM 1-1453 SIGNAL STATUS VALVE 47 NOT OK
AND T_ALARM_1_1453  ; ALARM 1-1453 SIGNAL STATUS VALVE 47 NOT OK
SET M_ALARM_1_1453  ; ALARM 1-1453 SIGNAL STATUS VALVE 47 NOT OK

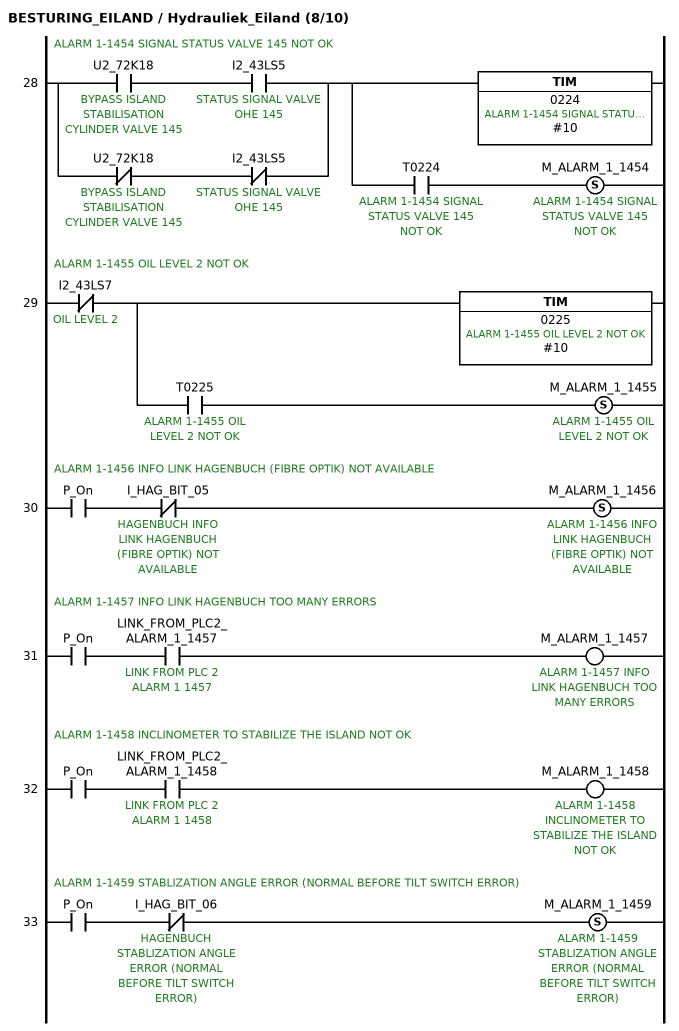
; rung 28: ALARM 1-1454 SIGNAL STATUS VALVE 145 NOT OK
LD U2_72K18  ; BYPASS ISLAND STABILISATION CYLINDER VALVE 145
AND I2_43LS5  ; STATUS SIGNAL VALVE OHE 145
LDNOT U2_72K18  ; BYPASS ISLAND STABILISATION CYLINDER VALVE 145
ANDNOT I2_43LS5  ; STATUS SIGNAL VALVE OHE 145
ORLD
TIM 0224 #10  ; ALARM 1-1454 SIGNAL STATUS VALVE 145 NOT OK
AND T0224  ; ALARM 1-1454 SIGNAL STATUS VALVE 145 NOT OK
SET M_ALARM_1_1454  ; ALARM 1-1454 SIGNAL STATUS VALVE 145 NOT OK
; rung 29: ALARM 1-1455 OIL LEVEL 2 NOT OK
LDNOT I2_43LS7  ; OIL LEVEL 2
TIM 0225 #10  ; ALARM 1-1455 OIL LEVEL 2 NOT OK
AND T0225  ; ALARM 1-1455 OIL LEVEL 2 NOT OK
SET M_ALARM_1_1455  ; ALARM 1-1455 OIL LEVEL 2 NOT OK
; rung 30: ALARM 1-1456 INFO LINK HAGENBUCH (FIBRE OPTIK) NOT AVAILABLE
LD P_On
ANDNOT I_HAG_BIT_05  ; HAGENBUCH INFO LINK HAGENBUCH (FIBRE OPTIK) NOT AVAILABLE
SET M_ALARM_1_1456  ; ALARM 1-1456 INFO LINK HAGENBUCH (FIBRE OPTIK) NOT AVAILABLE
; rung 31: ALARM 1-1457 INFO LINK HAGENBUCH TOO MANY ERRORS
LD P_On
AND LINK_FROM_PLC2_ALARM_1_1457  ; LINK FROM PLC 2 ALARM 1 1457
OUT M_ALARM_1_1457  ; ALARM 1-1457 INFO LINK HAGENBUCH TOO MANY ERRORS
; rung 32: ALARM 1-1458 INCLINOMETER TO STABILIZE THE ISLAND NOT OK
LD P_On
AND LINK_FROM_PLC2_ALARM_1_1458  ; LINK FROM PLC 2 ALARM 1 1458
OUT M_ALARM_1_1458  ; ALARM 1-1458 INCLINOMETER TO STABILIZE THE ISLAND NOT OK
; rung 33: ALARM 1-1459 STABLIZATION ANGLE ERROR (NORMAL BEFORE TILT SWITCH ERROR)
LD P_On
ANDNOT I_HAG_BIT_06  ; HAGENBUCH STABLIZATION ANGLE ERROR (NORMAL BEFORE TILT SWITCH ERROR)
SET M_ALARM_1_1459  ; ALARM 1-1459 STABLIZATION ANGLE ERROR (NORMAL BEFORE TILT SWITCH ERROR)

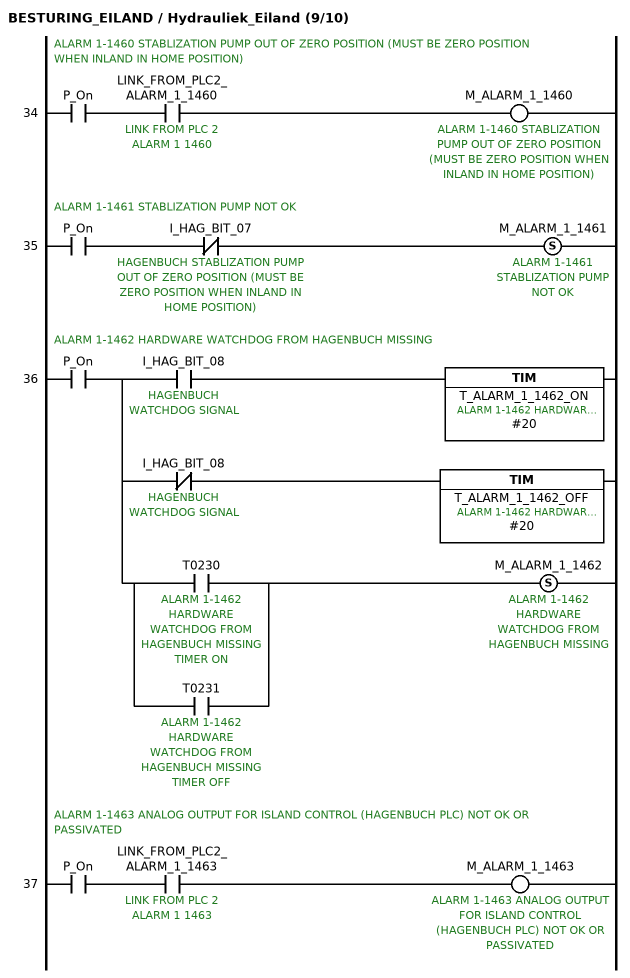
; rung 34: ALARM 1-1460 STABLIZATION PUMP OUT OF ZERO POSITION (MUST BE ZERO POSITION WHEN INLAND IN HOME POSITION)
LD P_On
AND LINK_FROM_PLC2_ALARM_1_1460  ; LINK FROM PLC 2 ALARM 1 1460
OUT M_ALARM_1_1460  ; ALARM 1-1460 STABLIZATION PUMP OUT OF ZERO POSITION (MUST BE ZERO POSITION WHEN INLAND IN HOME POSITION)
; rung 35: ALARM 1-1461 STABLIZATION PUMP NOT OK
LD P_On
ANDNOT I_HAG_BIT_07  ; HAGENBUCH STABLIZATION PUMP OUT OF ZERO POSITION (MUST BE ZERO POSITION WHEN INLAND IN HOME POSITION)
SET M_ALARM_1_1461  ; ALARM 1-1461 STABLIZATION PUMP NOT OK
; rung 36: ALARM 1-1462 HARDWARE WATCHDOG FROM HAGENBUCH MISSING
LD P_On
OUT TR0
AND I_HAG_BIT_08  ; HAGENBUCH WATCHDOG SIGNAL
TIM T_ALARM_1_1462_ON #20  ; ALARM 1-1462 HARDWARE WATCHDOG FROM HAGENBUCH MISSING TIMER ON
LD TR0
ANDNOT I_HAG_BIT_08  ; HAGENBUCH WATCHDOG SIGNAL
TIM T_ALARM_1_1462_OFF #20  ; ALARM 1-1462 HARDWARE WATCHDOG FROM HAGENBUCH MISSING TIMER OFF
LD TR0
LD T0230  ; ALARM 1-1462 HARDWARE WATCHDOG FROM HAGENBUCH MISSING TIMER ON
OR T0231  ; ALARM 1-1462 HARDWARE WATCHDOG FROM HAGENBUCH MISSING TIMER OFF
ANDLD
SET M_ALARM_1_1462  ; ALARM 1-1462 HARDWARE WATCHDOG FROM HAGENBUCH MISSING
; rung 37: ALARM 1-1463 ANALOG OUTPUT FOR ISLAND CONTROL (HAGENBUCH PLC) NOT OK OR PASSIVATED
LD P_On
AND LINK_FROM_PLC2_ALARM_1_1463  ; LINK FROM PLC 2 ALARM 1 1463
OUT M_ALARM_1_1463  ; ALARM 1-1463 ANALOG OUTPUT FOR ISLAND CONTROL (HAGENBUCH PLC) NOT OK OR PASSIVATED

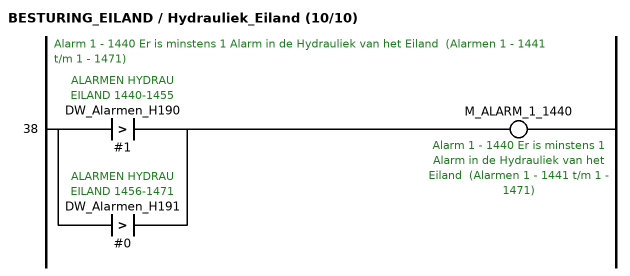
; rung 38: Alarm 1 - 1440 Er is minstens 1 Alarm in de Hydrauliek van het Eiland  (Alarmen 1 - 1441 t/m 1 - 1471)
LD>(320) DW_Alarmen_H190 #1  ; ALARMEN HYDRAU EILAND 1440-1455
OR>(320) DW_Alarmen_H191 #0  ; ALARMEN HYDRAU EILAND 1456-1471
OUT M_ALARM_1_1440  ; Alarm 1 - 1440 Er is minstens 1 Alarm in de Hydrauliek van het Eiland  (Alarmen 1 - 1441 t/m 1 - 1471)

### Section Stabilisatie_Eiland

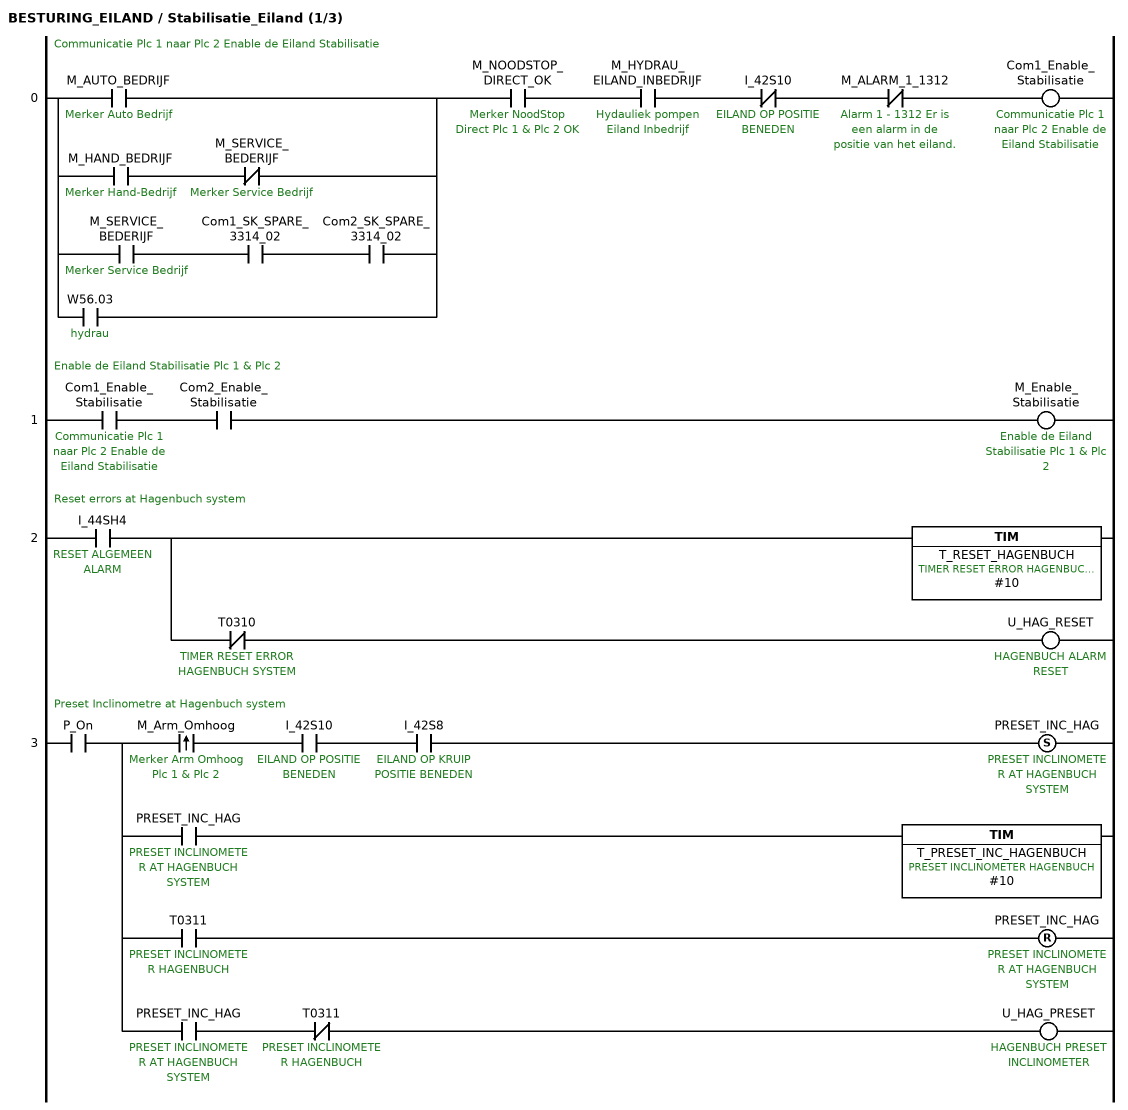
; rung 0: Communicatie Plc 1 naar Plc 2 Enable de Eiland Stabilisatie
LD M_AUTO_BEDRIJF  ; Merker Auto Bedrijf
LD M_HAND_BEDRIJF  ; Merker Hand-Bedrijf
ANDNOT M_SERVICE_BEDERIJF  ; Merker Service Bedrijf
ORLD
LD M_SERVICE_BEDERIJF  ; Merker Service Bedrijf
AND Com1_SK_SPARE_3314_02
AND Com2_SK_SPARE_3314_02
ORLD
OR W56.03  ; hydrau
AND M_NOODSTOP_DIRECT_OK  ; Merker NoodStop Direct Plc 1 & Plc 2 OK
AND M_HYDRAU_EILAND_INBEDRIJF  ; Hydauliek pompen Eiland Inbedrijf
ANDNOT I_42S10  ; EILAND OP POSITIE BENEDEN
ANDNOT M_ALARM_1_1312  ; Alarm 1 - 1312 Er is een alarm in de positie van het eiland.
OUT Com1_Enable_Stabilisatie  ; Communicatie Plc 1 naar Plc 2 Enable de Eiland Stabilisatie
; rung 1: Enable de Eiland Stabilisatie Plc 1 & Plc 2
LD Com1_Enable_Stabilisatie  ; Communicatie Plc 1 naar Plc 2 Enable de Eiland Stabilisatie
AND Com2_Enable_Stabilisatie
OUT M_Enable_Stabilisatie  ; Enable de Eiland Stabilisatie Plc 1 & Plc 2
; rung 2: Reset errors at Hagenbuch system
LD I_44SH4  ; RESET ALGEMEEN ALARM
TIM T_RESET_HAGENBUCH #10  ; TIMER RESET ERROR HAGENBUCH SYSTEM
ANDNOT T0310  ; TIMER RESET ERROR HAGENBUCH SYSTEM
OUT U_HAG_RESET  ; HAGENBUCH ALARM RESET
; rung 3: Preset Inclinometre at Hagenbuch system
LD P_On
OUT TR0
@AND M_Arm_Omhoog  ; Merker Arm Omhoog Plc 1 & Plc 2
AND I_42S10  ; EILAND OP POSITIE BENEDEN
AND I_42S8  ; EILAND OP KRUIP POSITIE BENEDEN
SET PRESET_INC_HAG  ; PRESET INCLINOMETER AT HAGENBUCH SYSTEM
LD TR0
AND PRESET_INC_HAG  ; PRESET INCLINOMETER AT HAGENBUCH SYSTEM
TIM T_PRESET_INC_HAGENBUCH #10  ; PRESET INCLINOMETER HAGENBUCH
LD TR0
AND T0311  ; PRESET INCLINOMETER HAGENBUCH
RSET PRESET_INC_HAG  ; PRESET INCLINOMETER AT HAGENBUCH SYSTEM
LD TR0
AND PRESET_INC_HAG  ; PRESET INCLINOMETER AT HAGENBUCH SYSTEM
ANDNOT T0311  ; PRESET INCLINOMETER HAGENBUCH
OUT U_HAG_PRESET  ; HAGENBUCH PRESET INCLINOMETER

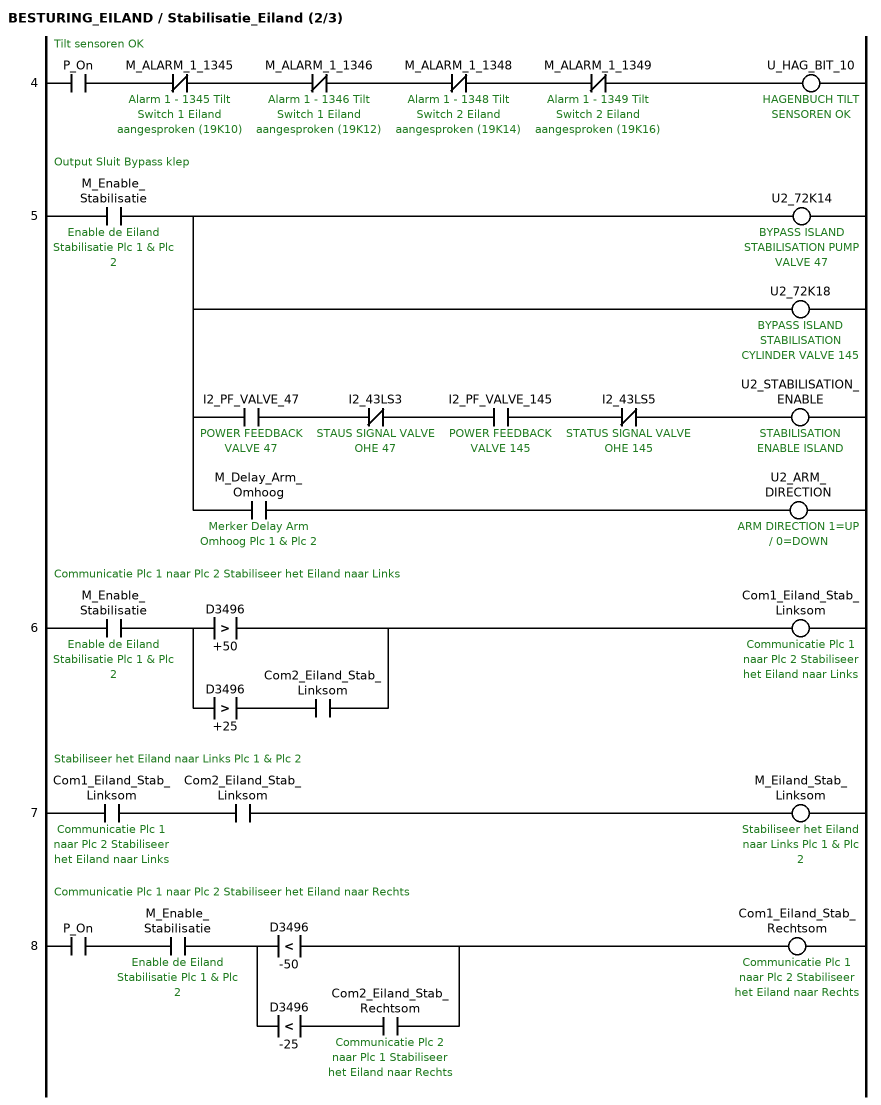
; rung 4: Tilt sensoren OK
LD P_On
ANDNOT M_ALARM_1_1345  ; Alarm 1 - 1345 Tilt Switch 1 Eiland aangesproken (19K10)
ANDNOT M_ALARM_1_1346  ; Alarm 1 - 1346 Tilt Switch 1 Eiland aangesproken (19K12)
ANDNOT M_ALARM_1_1348  ; Alarm 1 - 1348 Tilt Switch 2 Eiland aangesproken (19K14)
ANDNOT M_ALARM_1_1349  ; Alarm 1 - 1349 Tilt Switch 2 Eiland aangesproken (19K16)
OUT U_HAG_BIT_10  ; HAGENBUCH TILT SENSOREN OK
; rung 5: Output Sluit Bypass klep
LD M_Enable_Stabilisatie  ; Enable de Eiland Stabilisatie Plc 1 & Plc 2
OUT TR0
OUT U2_72K14  ; BYPASS ISLAND STABILISATION PUMP VALVE 47
OUT U2_72K18  ; BYPASS ISLAND STABILISATION CYLINDER VALVE 145
AND I2_PF_VALVE_47  ; POWER FEEDBACK VALVE 47
ANDNOT I2_43LS3  ; STAUS SIGNAL VALVE OHE 47
AND I2_PF_VALVE_145  ; POWER FEEDBACK VALVE 145
ANDNOT I2_43LS5  ; STATUS SIGNAL VALVE OHE 145
OUT U2_STABILISATION_ENABLE  ; STABILISATION ENABLE ISLAND
LD TR0
AND M_Delay_Arm_Omhoog  ; Merker Delay Arm Omhoog Plc 1 & Plc 2
OUT U2_ARM_DIRECTION  ; ARM DIRECTION 1=UP / 0=DOWN
; rung 6: Communicatie Plc 1 naar Plc 2 Stabiliseer het Eiland naar Links
LD M_Enable_Stabilisatie  ; Enable de Eiland Stabilisatie Plc 1 & Plc 2
LD>S(322) D3496 +50
LD>S(322) D3496 +25
AND Com2_Eiland_Stab_Linksom
ORLD
ANDLD
OUT Com1_Eiland_Stab_Linksom  ; Communicatie Plc 1 naar Plc 2 Stabiliseer het Eiland naar Links
; rung 7: Stabiliseer het Eiland naar Links Plc 1 & Plc 2
LD Com1_Eiland_Stab_Linksom  ; Communicatie Plc 1 naar Plc 2 Stabiliseer het Eiland naar Links
AND Com2_Eiland_Stab_Linksom
OUT M_Eiland_Stab_Linksom  ; Stabiliseer het Eiland naar Links Plc 1 & Plc 2
; rung 8: Communicatie Plc 1 naar Plc 2 Stabiliseer het Eiland naar Rechts
LD P_On
AND M_Enable_Stabilisatie  ; Enable de Eiland Stabilisatie Plc 1 & Plc 2
LD<S(312) D3496 -50
LD<S(312) D3496 -25
AND Com2_Eiland_Stab_Rechtsom  ; Communicatie Plc 2 naar Plc 1 Stabiliseer het Eiland naar Rechts
ORLD
ANDLD
OUT Com1_Eiland_Stab_Rechtsom  ; Communicatie Plc 1 naar Plc 2 Stabiliseer het Eiland naar Rechts

